// Startup hook called after PreInit and Init.
INTERFACE I_PostInit EXTENDS I_Generic

// Called once during Plant startup after Init.
METHOD PostInit
END_METHOD

END_INTERFACE

(* stored: Version 1.1.0.1
   Itf I_PostInit: Id {9b9651e4-045e-4b17-8f2b-108f12ea7bf1}
   Method PostInit: Id {1237434a-0b74-4202-8a56-33e757a0a879} *)
